FUNCTION_BLOCK FB_Homing
VAR_IN_OUT
    AxisRef: AXIS_REF;
	
END_VAR
VAR_INPUT
    bExecute: BOOL;
    bLimitFwd: BOOL;
    bLimitBwd: BOOL;
    bHomeSensor: BOOL;
    eHomeSeq: E_HomingRoutines;
    fHomePosition: LREAL;
    fHomeFinishDistance: LREAL;
	fHomeAbsPosition : LREAL;
	bDoAbsoluteMove : BOOL;
	fHomeMidRelativeMove : LREAL;
    stConfig: ST_AxisConfig;
	stHomingConfig : ST_AxisHomingConfig;
	bGoToFwdLimitFirst : BOOL;
	bGoToBwdLimitFirst : BOOL;
	fFastVelocity : LREAL;
END_VAR
VAR_OUTPUT
    bDone : BOOL;
    bBusy: BOOL;
    bCommandAborted: BOOL;
    bError: BOOL;
    nErrorId: UDINT;
	bInHomingSequence: BOOL;
END_VAR
VAR
    //Beckhoff homing function blocks
    fbStepLimitSwitchPreparation: MC_StepLimitSwitchDetection;
    fbStepLimitSwitchDetection: MC_StepLimitSwitchDetection;
    fbStepAbsoluteSwitchDetection: MC_StepAbsoluteSwitchDetection;
	fbStepAbsoluteSwitchPreparation: MC_StepAbsoluteSwitchDetection;
	fbStepReferencePulsePreparation: MC_StepReferencePulseDetection;
    fbStepReferencePulseDetection: MC_StepReferencePulseDetection;
    fbStepBlockLagDetection: MC_StepBlockLagBasedDetection;
    fbHomeDirect: MC_HomeDirect;
    fbSetPos: MC_SetPosition;
    fbFinishHoming: MC_FinishHoming;
    fbAbortHoming: MC_AbortHoming;
	fbMoveRelative : MC_MoveRelative;
	fbMoveAbsolute : MC_MoveAbsolute;
	fbMoveVelocity : MC_MoveVelocity;
    //Hardware Signals
    eLimitSwitchMode: MC_Switch_Mode := mcRisingEdge;
    stLimitSwitchSignal: MC_Ref_Signal_Ref;
    eRefSwitchMode: MC_Switch_Mode := mcRisingEdge;
    stRefSwitchSignal: MC_Ref_Signal_Ref;
    stEncPulseSignal: MC_Ref_Signal_Ref;
    //Homing parameters
    stPreparationDirection: MC_Home_Direction;
    stDetectDirection: MC_Home_Direction;
    stHomingParameter: MC_HomingParameter;
    stOptions: ST_Home_Options4;
    stOptions3: ST_Home_Options3;
    fbVelocityToCam: MC_ReadParameter;
    fVelocityToCam: LREAL;
    fbVelocityFromCam: MC_ReadParameter;
    fVelocityFromCam: LREAL;
    //State machine
    fbExecute: R_TRIG;
    bViaLimitSwitch: BOOL;
	bViaFastEncPulse : BOOL;
	bViaFastRef : BOOL;
    eHomingState: (eWaitForRequest := 0, ePreparation := 1, eDetection := 2, eSetPos := 3, eFinishHoming := 4, eMoveRelative:=5, eAbsMove:=6, eAbortHoming := 20, eGoToFwd:=7, eGoToBwd:=8, eWaitForFwd:=9,eWaitForBwd:=10);
    iErrorId: UDINT;
    bDetectionFB_Execute: BOOL;
    bDetectionFB_Done: BOOL;
    bDetectionFB_Busy: BOOL;
    bDetectionFB_CommandAborted: BOOL;
    bDetectionFB_Error: BOOL;
    nDetectionFB_ErrorID: UDINT;
    fRecordedPosition: LREAL;
    fRecordedPositionLatched: LREAL;
END_VAR

bInHomingSequence:= FALSE;
//Hardware signals
stLimitSwitchSignal.SignalSource := SignalSource_Default;
stLimitSwitchSignal.TouchProbe := PlcEvent;
stRefSwitchSignal.SignalSource := SignalSource_Default;
stRefSwitchSignal.TouchProbe := PlcEvent;
stRefSwitchSignal.Level := bHomeSensor;
stEncPulseSignal.SignalSource := SignalSource_ZeroPulse;
stEncPulseSignal.TouchProbe := TouchProbe1;

fbMoveRelative(
	Axis:= AxisRef, Velocity:= fVelocityToCam);
	fbMoveRelative.Execute:= FALSE;

fbMoveAbsolute(
	Axis:= AxisRef, Velocity:= fFastVelocity, Position:= fHomeAbsPosition);
	fbMoveAbsolute.Execute:= FALSE;

//Constantly read the NC for homing velocities so they are available when a homing is executed
fbVelocityToCam(
    Axis := AxisRef,
    Enable := TRUE,
    ParameterNumber := E_AxisParameters.AxisVelocityToCam,
    ReadMode := READMODE_CYCLIC);

fbVelocityFromCam(
    Axis := AxisRef,
    Enable := TRUE,
    ParameterNumber := E_AxisParameters.AxisVelocityFromCam,
    ReadMode := READMODE_CYCLIC);

    //Only write velocity if the function block has not errored
IF NOT fbVelocityToCam.Error THEN
    fVelocityToCam := fbVelocityToCam.Value;
END_IF

IF NOT fbVelocityFromCam.Error THEN
    fVelocityFromCam := fbVelocityFromCam.Value;
END_IF

    //Feeds function block errors through
IF fbVelocityToCam.Error THEN
    bError := TRUE;
    nErrorID := fbVelocityToCam.ErrorID;

ELSIF fbVelocityFromCam.Error THEN
    bError := TRUE;
    nErrorID := fbVelocityFromCam.ErrorID;
END_IF

//Common function blocks used for all routines
stOptions.DisableDriveAccess := stHomingConfig.bDisableDriveAccess;

//For StepBlockLagDetection
stOptions3.DisableDriveAccess := stHomingConfig.bDisableDriveAccess;

fbStepLimitSwitchPreparation.Options.DisableDriveAccess := stOptions.DisableDriveAccess;
fbStepLimitSwitchPreparation(
    Axis := AxisRef,
    Parameter := stHomingParameter,
    Direction := stPreparationDirection,
    LimitSwitchMode:= eLimitSwitchMode,
    LimitSwitchSignal:= stLimitSwitchSignal,
    Velocity := fVelocityToCam);
	


fbSetPos(
    Axis := AxisRef,
    Position := AxisRef.NcToPlc.ActPos - fRecordedPositionLatched + fHomePosition);

fbFinishHoming.Options.DisableDriveAccess := stOptions.DisableDriveAccess;
fbFinishHoming(
    Axis := AxisRef,
    Parameter := stHomingParameter,
    Velocity := fVelocityFromCam);

fbMoveVelocity(Axis:= AxisRef, Velocity:= ABS(fFastVelocity));
	fbMoveVelocity.Execute:= FALSE;

fbAbortHoming.Options.DisableDriveAccess := stOptions.DisableDriveAccess;
fbAbortHoming(
    Axis := AxisRef,
    Parameter := stHomingParameter);

//ACTs contain function blocks custom to each individual routine for the detection stage
CASE eHomeSeq OF
    E_HomingRoutines.eHomeToLimit_Bwd,
    E_HomingRoutines.eHomeToLimit_Fwd:
        actHomeToLimit();

    E_HomingRoutines.eHomeToRef_Bwd,
	E_HomingRoutines.eHomeToRef_Bwd_Fast,
	E_HomingRoutines.eHomeToRef_Fwd_Fast,
    E_HomingRoutines.eHomeToRef_Fwd:
        actHomeToRef();

    E_HomingRoutines.eHomeToEncPulse_Bwd,
    E_HomingRoutines.eHomeToEncPulse_Fwd,
    E_HomingRoutines.eHomeToEncPulse_viaBwdLimit,
    E_HomingRoutines.eHomeToEncPulse_viaFwdLimit,
	E_HomingRoutines.eHomeToEncPulse_BWD_FAST,
	E_HomingRoutines.eHomeToEncPulse_FWD_FAST:
        actHomeToEncPulse();

    E_HomingRoutines.eHomeToBlock_Bwd,
    E_HomingRoutines.eHomeToBlock_Fwd:
        actHomeToBlock();

    E_HomingRoutines.eHomeDirect:
        actHomeDirect();
END_CASE


//State machine
fbExecute(CLK:= bExecute);
CASE eHomingState OF

    eWaitForRequest:
        IF NOT bExecute THEN
            bBusy := FALSE;
            bDone := FALSE;
            bCommandAborted := FALSE;
            bError := FALSE;
            nErrorID := 0;
            iErrorID := 0;

            fbStepLimitSwitchPreparation.Execute := FALSE;
            fbStepLimitSwitchDetection.Execute := FALSE;
            fbStepAbsoluteSwitchDetection.Execute := FALSE;
			fbStepReferencePulsePreparation.Execute := FALSE;
            fbStepReferencePulseDetection.Execute := FALSE;
            fbStepBlockLagDetection.Execute := FALSE;
            fbHomeDirect.Execute := FALSE;
            fbSetPos.Execute := FALSE;
            fbFinishHoming.Execute := FALSE;
            fbAbortHoming.Execute := FALSE;
        END_IF

        IF fbExecute.Q AND NOT(eHomeSeq = E_HomingRoutines.eNoHoming)THEN
            bBusy:= TRUE;
			IF bGoToFwdLimitFirst THEN
				eHomingState:= eGoToFwd;
			ELSIF bGoToBwdLimitFirst THEN
				eHomingState:= eGoToBwd;
			ELSE
				eHomingState:= ePreparation;
			END_IF            
        END_IF

	eGoToFwd:
		fbMoveVelocity.Execute:= TRUE;
		fbMoveVelocity.Direction:= MC_Direction.MC_Positive_Direction;
		eHomingState:= eWaitForFwd;
		bInHomingSequence:= TRUE;
		
	eWaitForFwd:
		IF NOT bLimitFwd THEN
			eHomingState:= ePreparation;
		END_IF
		bInHomingSequence:= TRUE;
		//IF NOT fbMoveVelocity.Active THEN
		//	eHomingState:= eAbortHoming;
		//END_IF
		
	eGoToBwd:
		fbMoveVelocity.Direction:= MC_Direction.MC_Negative_Direction;
		fbMoveVelocity.Execute:= TRUE;
		eHomingState:= eWaitForBwd;
		bInHomingSequence:= TRUE;
		
	eWaitForBwd:
		IF NOT bLimitBwd THEN
			eHomingState:= ePreparation;
		END_IF
		bInHomingSequence:= TRUE;
		//IF NOT fbMoveVelocity.Active THEN
		//	eHomingState:= eAbortHoming;
		//END_IF

    ePreparation: //If bViaLimitSwitch is set TRUE then go first to a limit otherwise skip this step
		bInHomingSequence:= TRUE;
        IF bViaLimitSwitch THEN
            fbStepLimitSwitchPreparation.Execute := TRUE;
        ELSIF bViaFastEncPulse THEN
			fbStepReferencePulsePreparation.Execute := TRUE;
		ELSIF bViaFastRef THEN
			fbStepAbsoluteSwitchPreparation.Execute:= TRUE;
		ELSE
            eHomingState := eDetection;
        END_IF

		IF bViaLimitSwitch THEN
        	IF NOT fbStepLimitSwitchPreparation.Busy AND fbStepLimitSwitchPreparation.Done THEN
            	fbStepLimitSwitchPreparation.Execute := FALSE;
            	eHomingState := eDetection;
        	ELSIF NOT fbStepLimitSwitchPreparation.Busy AND (fbStepLimitSwitchPreparation.Error OR fbStepLimitSwitchPreparation.CommandAborted) THEN
            	iErrorID := fbStepLimitSwitchPreparation.ErrorID;
            	fbStepLimitSwitchPreparation.Execute := FALSE;
            	eHomingState := eAbortHoming;
        	END_IF
		END_IF
		IF bViaFastEncPulse THEN
			IF NOT fbStepReferencePulsePreparation.Busy AND fbStepReferencePulsePreparation.Done THEN
            	fbStepReferencePulsePreparation.Execute := FALSE;
            	eHomingState := eMoveRelative;
        	ELSIF NOT fbStepReferencePulsePreparation.Busy AND (fbStepReferencePulsePreparation.Error OR fbStepReferencePulsePreparation.CommandAborted) THEN
            	iErrorID := fbStepReferencePulsePreparation.ErrorID;
            	fbStepReferencePulsePreparation.Execute := FALSE;
            	eHomingState := eAbortHoming;
        	END_IF			
		END_IF
		IF bViaFastRef THEN
			IF NOT fbStepAbsoluteSwitchPreparation.Busy AND fbStepAbsoluteSwitchPreparation.Done THEN
            	fbStepAbsoluteSwitchPreparation.Execute := FALSE;
            	eHomingState := eMoveRelative;
        	ELSIF NOT fbStepAbsoluteSwitchPreparation.Busy AND (fbStepAbsoluteSwitchPreparation.Error OR fbStepAbsoluteSwitchPreparation.CommandAborted) THEN
            	iErrorID := fbStepAbsoluteSwitchPreparation.ErrorID;
            	fbStepAbsoluteSwitchPreparation.Execute := FALSE;
            	eHomingState := eAbortHoming;
        	END_IF			
		END_IF
		
	eMoveRelative:
		bInHomingSequence:= TRUE;
		fbMoveRelative.Execute:= TRUE;
		IF NOT fbMoveRelative.Busy AND fbMoveRelative.Done THEN
            	fbMoveRelative.Execute := FALSE;
            	eHomingState := eDetection;
        	ELSIF NOT fbMoveRelative.Busy AND (fbMoveRelative.Error OR fbMoveRelative.CommandAborted) THEN
            	iErrorID := fbMoveRelative.ErrorID;
            	fbMoveRelative.Execute := FALSE;
            	eHomingState := eAbortHoming;
        	END_IF


    eDetection: //Use bDetectionFB_<BOOL Variables> to interact with different detection FBs located in ACTs
		bInHomingSequence:= FALSE;
        bDetectionFB_Execute := TRUE;

        IF NOT bDetectionFB_Busy AND bDetectionFB_Done THEN
            bDetectionFB_Execute := FALSE;
            fRecordedPositionLatched := fRecordedPosition;
            IF eHomeSeq = E_HomingRoutines.eHomeDirect THEN
                bBusy := fbHomeDirect.Busy;
                bDone := fbHomeDirect.Done;
                bCommandAborted := fbHomeDirect.CommandAborted;
                bError := fbHomeDirect.Error;
                nErrorId := fbHomeDirect.ErrorID;
                eHomingState := eWaitForRequest;
            ELSE
                eHomingState := eSetPos;
            END_IF
        ELSIF NOT bDetectionFB_Busy AND (bDetectionFB_Error OR bDetectionFB_CommandAborted) THEN
            iErrorID := nDetectionFB_ErrorID;
            bDetectionFB_Execute := FALSE;
            eHomingState := eAbortHoming;
        END_IF


    eSetPos:
		bInHomingSequence:= FALSE;
        fbSetPos.Execute := TRUE;

        fbSetPos.Options.ClearPositionLag := TRUE;
        IF NOT fbSetPos.Busy AND fbSetPos.Done THEN
            fbSetPos.Execute := FALSE;
			IF bDoAbsoluteMove THEN
				eHomingState := eAbsMove;
			ELSE
				 eHomingState := eFinishHoming;
			END_IF
			
           
        ELSIF NOT fbSetPos.Busy AND fbSetPos.Error THEN
            iErrorID := fbSetPos.ErrorID;
            fbSetPos.Execute := FALSE;
            eHomingState := eAbortHoming;
        END_IF
	
	eAbsMove:
		bInHomingSequence:= FALSE;
		fbMoveAbsolute.Execute:= TRUE;
		IF NOT fbMoveAbsolute.Busy AND fbMoveAbsolute.Done THEN
            fbMoveAbsolute.Execute := FALSE;
            eHomingState := eFinishHoming;
        ELSIF NOT fbMoveAbsolute.Busy AND (fbMoveAbsolute.Error OR fbMoveAbsolute.CommandAborted) THEN
            iErrorID := fbMoveAbsolute.ErrorID;
            fbMoveAbsolute.Execute := FALSE;
            eHomingState := eAbortHoming;
        END_IF

    eFinishHoming:
		bInHomingSequence:= FALSE;
        fbFinishHoming.Execute := TRUE;

        IF NOT fbFinishHoming.Busy AND fbFinishHoming.Done THEN
            bBusy := FALSE;
            bDone := TRUE;
            fbFinishHoming.Execute := FALSE;
            eHomingState := eWaitForRequest;
        ELSIF NOT fbFinishHoming.Busy AND (fbFinishHoming.Error OR fbFinishHoming.CommandAborted) THEN
            iErrorID := fbFinishHoming.ErrorID;
            fbFinishHoming.Execute := FALSE;
            eHomingState := eAbortHoming;
        END_IF


    eAbortHoming:
		bInHomingSequence:= FALSE;
        fbAbortHoming.Execute := TRUE;

        IF NOT fbAbortHoming.Busy AND fbAbortHoming.Done THEN
            bBusy := FALSE;
            IF iErrorId <> 0 THEN
                bError := TRUE;
                nErrorId := iErrorId;
            ELSE
                bCommandAborted := TRUE;
            END_IF
            fbAbortHoming.Execute := FALSE;
            eHomingState := eWaitForRequest;
        ELSIF NOT fbAbortHoming.Busy AND fbAbortHoming.Error THEN
            bBusy := FALSE;
            bError := TRUE;
            nErrorID := fbAbortHoming.ErrorID;
            fbAbortHoming.Execute := FALSE;
            eHomingState := eWaitForRequest;
        END_IF

END_CASE

ACTION actHomeDirect:

bViaLimitSwitch := FALSE;

fbHomeDirect(
    Axis := AxisRef,
    Parameter := stHomingParameter,
    Execute := bDetectionFB_Execute,
    SetPosition := fHomePosition,
    Done => bDetectionFB_Done,
    Busy => bDetectionFB_Busy,
    CommandAborted => bDetectionFB_CommandAborted,
    Error => bDetectionFB_Error,
    ErrorID => nDetectionFB_ErrorID);
END_ACTION

ACTION actHomeToBlock:
CASE eHomeSeq OF
    E_HomingRoutines.eHomeToBlock_Bwd:
        stDetectDirection:= mcNegativeDirection;
        fbFinishHoming.Distance := fHomeFinishDistance;
    E_HomingRoutines.eHomeToBlock_Fwd:
        stDetectDirection:= mcPositiveDirection;
        fbFinishHoming.Distance := -fHomeFinishDistance;
END_CASE

bViaLimitSwitch:=FALSE;

fbStepBlockLagDetection(
    Axis := AxisRef,
    Execute := bDetectionFB_Execute,
    Parameter := stHomingParameter,
    Direction := stDetectDirection,
    Velocity := fVelocityFromCam, //Maximum travel velocity (>0).
    DetectionVelocityLimit := stHomingConfig.fDetectionVelocityLimit, //Velocity that must be fallen below for the time DetectionVelocityTime in order to detect driving against the fixed stop.
    DetectionVelocityTime := stHomingConfig.tDetectionVelocityTime, //Time for detecting the velocity undershoot when driving against the fixed stop.
    TimeLimit :=  stHomingConfig.tTimeLimit, //Exceeding this time leads to the search procedure being aborted.
    DistanceLimit := stHomingConfig.fDistanceLimit, //Exceeding this distance in relation to the start position leads to the search procedure being aborted.
    TorqueLimit := stHomingConfig.fTorqueLimit, //The motor torque is limited to this value (percentage of configured channel peak torque), in relation to the weight counterbalance that is possibly parameterized in the drive, in order to avoid mechanical damage.
    LagLimit := stHomingConfig.fLagLimit, //Position lag value which, if exceeded, leads to detection of driving against the fixed stop.
    Options := stOptions3,
    Done => bDetectionFB_Done,
    Busy => bDetectionFB_Busy,
    CommandAborted => bDetectionFB_CommandAborted,
    Error => bDetectionFB_Error,
    ErrorID => nDetectionFB_ErrorID,
    RecordedPosition => fRecordedPosition);
END_ACTION

ACTION actHomeToEncPulse:

CASE eHomeSeq OF
    E_HomingRoutines.eHomeToEncPulse_Bwd:
        stDetectDirection := mcNegativeDirection;
        fbFinishHoming.Distance := fHomeFinishDistance;
        bViaLimitSwitch := FALSE;
		bViaFastEncPulse:= FALSE;
		bViaFastRef := FALSE;
    E_HomingRoutines.eHomeToEncPulse_Fwd:
        stDetectDirection := mcPositiveDirection;
        fbFinishHoming.Distance := -fHomeFinishDistance;
        bViaLimitSwitch := FALSE;
		bViaFastEncPulse:= FALSE;
		bViaFastRef := FALSE;
    E_HomingRoutines.eHomeToEncPulse_viaBwdLimit:
        stDetectDirection := mcPositiveDirection;
        fbFinishHoming.Distance := fHomeFinishDistance;
        stPreparationDirection := mcNegativeDirection;
        stLimitSwitchSignal.Level := NOT(bLimitBwd);
        bViaLimitSwitch := TRUE;
		bViaFastEncPulse:= FALSE;
		bViaFastRef := FALSE;
    E_HomingRoutines.eHomeToEncPulse_viaFwdLimit:
        stDetectDirection := mcNegativeDirection;
        fbFinishHoming.Distance := -fHomeFinishDistance;
        stPreparationDirection := mcPositiveDirection;
        stLimitSwitchSignal.Level := NOT(bLimitFwd);
        bViaLimitSwitch := TRUE;
		bViaFastEncPulse:= FALSE;
		bViaFastRef := FALSE;
	
	E_HomingRoutines.eHomeToEncPulse_BWD_FAST:
		stDetectDirection := mcNegativeDirection;
        fbFinishHoming.Distance := fHomeFinishDistance;
        bViaLimitSwitch := FALSE;
		bViaFastEncPulse:= TRUE;
		bViaFastRef := FALSE;
		fbMoveRelative.Distance:= ABS(fHomeMidRelativeMove);
	
	E_HomingRoutines.eHomeToEncPulse_FWD_FAST:
		stDetectDirection := mcPositiveDirection;
        fbFinishHoming.Distance := fHomeFinishDistance;
        bViaLimitSwitch := FALSE;
		bViaFastEncPulse:= TRUE;
		fbMoveRelative.Distance:= -ABS(fHomeMidRelativeMove);
END_CASE

fbStepReferencePulsePreparation.Options.DisableDriveAccess := stOptions.DisableDriveAccess;
fbStepReferencePulsePreparation(
    Axis := AxisRef,
    Parameter := stHomingParameter,
    Direction := stDetectDirection,
    ReferenceSignal := stEncPulseSignal,
    Velocity := fVelocityToCam,
    Options := stOptions);
	

fbStepReferencePulseDetection.Options.DisableDriveAccess:= stOptions.DisableDriveAccess;
fbStepReferencePulseDetection(
    Axis := AxisRef,
    Execute := bDetectionFB_Execute,
    Parameter := stHomingParameter,
    Direction := stDetectDirection,
    ReferenceSignal := stEncPulseSignal,
    Velocity := fVelocityFromCam,
    Options := stOptions,
    Done => bDetectionFB_Done,
    Busy => bDetectionFB_Busy,
    CommandAborted => bDetectionFB_CommandAborted,
    Error => bDetectionFB_Error,
    ErrorID => nDetectionFB_ErrorID,
    RecordedPosition => fRecordedPosition);
END_ACTION

ACTION actHomeToLimit:

CASE eHomeSeq OF
    E_HomingRoutines.eHomeToLimit_Bwd:
        stLimitSwitchSignal.Level := NOT(bLimitBwd);
        stDetectDirection:= mcNegativeDirection;
        fbFinishHoming.Distance := fHomeFinishDistance;
    E_HomingRoutines.eHomeToLimit_Fwd:
        stLimitSwitchSignal.Level := NOT(bLimitFwd);
        stDetectDirection:= mcPositiveDirection;
        fbFinishHoming.Distance := -fHomeFinishDistance;
END_CASE
bViaLimitSwitch:=FALSE;

fbStepLimitSwitchDetection.Options.DisableDriveAccess:= stOptions.DisableDriveAccess;
fbStepLimitSwitchDetection(
    Axis := AxisRef,
    Execute := bDetectionFB_Execute,
    Parameter := stHomingParameter,
    Direction := stDetectDirection,
    LimitSwitchMode := eLimitSwitchMode,
    LimitSwitchSignal := stLimitSwitchSignal,
    Velocity := fVelocityFromCam,
    Options := stOptions,
    Done => bDetectionFB_Done,
    Busy => bDetectionFB_Busy,
    CommandAborted => bDetectionFB_CommandAborted,
    Error => bDetectionFB_Error,
    ErrorID => nDetectionFB_ErrorID,
    RecordedPosition => fRecordedPosition);
END_ACTION

ACTION actHomeToRef:

CASE eHomeSeq OF
    E_HomingRoutines.eHomeToRef_Bwd:
        stDetectDirection := mcNegativeDirection;
        fbFinishHoming.Distance := fHomeFinishDistance;
		bViaFastRef := FALSE;
		bViaLimitSwitch := FALSE;
		bViaFastEncPulse:= FALSE;
		
    E_HomingRoutines.eHomeToRef_Fwd:
        stDetectDirection := mcPositiveDirection;
        fbFinishHoming.Distance := -fHomeFinishDistance;
		bViaFastRef := FALSE;
		bViaLimitSwitch := FALSE;
		bViaFastEncPulse:= FALSE;
		
	E_HomingRoutines.eHomeToRef_Bwd_Fast:
        stDetectDirection := mcNegativeDirection;
        fbFinishHoming.Distance := fHomeFinishDistance;
		fbMoveRelative.Distance:= ABS(fHomeMidRelativeMove);
		bViaFastRef := TRUE;
		bViaLimitSwitch := FALSE;
		bViaFastEncPulse:= FALSE;
		
    E_HomingRoutines.eHomeToRef_Fwd_Fast:
        stDetectDirection := mcPositiveDirection;
        fbFinishHoming.Distance := -fHomeFinishDistance;
		fbMoveRelative.Distance:= -ABS(fHomeMidRelativeMove);
		bViaFastRef := TRUE;
		bViaLimitSwitch := FALSE;
		bViaFastEncPulse:= FALSE;
		
END_CASE
bViaLimitSwitch := FALSE;

fbStepAbsoluteSwitchDetection.Options.DisableDriveAccess := stOptions.DisableDriveAccess;
fbStepAbsoluteSwitchDetection(
    Axis := AxisRef,
    Execute := bDetectionFB_Execute,
    Parameter := stHomingParameter,
    Direction := stDetectDirection,
    SwitchMode := eRefSwitchMode,
    ReferenceSignal := stRefSwitchSignal,
    Velocity := fVelocityFromCam,
    PositiveLimitSwitch := NOT(bLimitFwd),
    NegativeLimitSwitch := NOT(bLimitBwd),
    Options := stOptions,
    Done => bDetectionFB_Done,
    Busy => bDetectionFB_Busy,
    CommandAborted => bDetectionFB_CommandAborted,
    Error => bDetectionFB_Error,
    ErrorID => nDetectionFB_ErrorID,
    RecordedPosition => fRecordedPosition);
	
fbStepAbsoluteSwitchPreparation.Options.DisableDriveAccess := stOptions.DisableDriveAccess;
fbStepAbsoluteSwitchPreparation(
    Axis := AxisRef,
    Parameter := stHomingParameter,
    Direction := stDetectDirection,
    SwitchMode := eRefSwitchMode,
    ReferenceSignal := stRefSwitchSignal,
    Velocity := fVelocityToCam,
    PositiveLimitSwitch := NOT(bLimitFwd),
    NegativeLimitSwitch := NOT(bLimitBwd),
    Options := stOptions);
END_ACTION

END_FUNCTION_BLOCK

(* stored: Version 1.1.0.1, ProductVersion 3.1.4026.18
   POU FB_Homing: Id {427b1d22-ef01-4bbb-ab89-ec8be67f3887}, SpecialFunc None
   Action actHomeDirect: Id {d23628f6-b24a-4bef-81d2-3d83fde8f1cd}
   Action actHomeToBlock: Id {7f7639d4-e566-498f-a828-fad9ed0e5d95}
   Action actHomeToEncPulse: Id {48b338da-ce35-49b7-b692-c1dd5d495b98}
   Action actHomeToLimit: Id {3859e05e-8699-4334-9196-1315e94174a0}
   Action actHomeToRef: Id {1a440701-e71d-439b-9045-d08d31798b28} *)
